// TIA Portal V20 export
TYPE "HMI_MotRevL"
   STRUCT
      FwdMan : Bool := FALSE;   // 1=Start: Forward Start Command in Manual Mode
      StopMan : Bool := FALSE;   // 1=Stop: Stop Command in Manual Mode
      RevMan : Bool := FALSE;   // 1=Start: Reverse Start Command in Manual Mode
      AutModOp : Bool := FALSE;   // 1=Auto Mode: Auto Mode by Operator
      ManModOp : Bool := TRUE;   // 1=Manual Mode: Manual Mode by Operator
      LocalLi : Bool;   // 1=Local Mode: Local Operation by Field Signal
      LocalOp : Bool := FALSE;   // 1=Local Mode: Local Operation by Operator
      OosOp : Bool := FALSE;   // 1=Oos Mode: Oos Mode by Operator
      FwdLocal : Bool;   // 1=Start Local: Field Forward Start Signal
      StopLocal : Bool;   // 1=Stop Local: Field Stop Signal
      RevLocal : Bool;   // 1=Start Local: Field Reverse Start Signal
      Monitor : Bool := TRUE;   // 1=Monitor ON, 0=Monitor OFF: Feedback Monitor
      MonTiStatic : Real := 3.0;   // Monitoring Time of Feedback [s]
      MonTiDynamic : Real := 3.0;   // Monitoring Time of Feedback on starting or on change in control output [s]
      MonTiDyStop : Real := 3.0;   // Monitoring Time of Feedback on stopping in control output [s]
      RapidStp : Bool := FALSE;   // 1 = Motor Rapid Stop command
      RstOp : Bool := FALSE;   // Operator Reset Signal
      Permit_ST : Byte := BYTE#16#FF;   // Permit Signal Status
      PermRev_ST : Byte := BYTE#16#FF;   // PermRev Signal Status
      Intlock_ST : Byte := BYTE#16#FF;   // Intlock Signal Status
      IntlRev_ST : Byte := BYTE#16#FF;   // IntlRev Signal Status
      Protect_ST : Byte := BYTE#16#FF;   // Protect Signal Status
      ProtRev_ST : Byte := BYTE#16#FF;   // ProtRev Signal Status
      UserAna1 : Real;   // User Analog Input 1
      UA1unit : Int := 0;   // Unit of UserAna1
      UserAna2 : Real;   // User Analog Input 2
      UA2unit : Int := 0;   // Unit of UserAna2
      BatchID : DWord := 16#0;   // Current Batch ID (number)
      BatchName : String[32] := '';   // Current Batch Name
      StepNo : DWord := 16#0;   // Batch Step Number
      CurrMon { ExternalWritable := 'False'} : DInt := 0;   // Remaining monitoring time [s]
      OS_PermOut { ExternalWritable := 'False'} : DWord := DWORD#16#FFFF_FFFF;   // Operator Permission: Output for OS
      OS_PermLog { ExternalWritable := 'False'} : DWord := DWORD#16#FFFF_FFFF;   // Operator Permission: Output for OS
      OpSt_Out { ExternalWritable := 'False'} : DWord := 16#0;   // Enabled operator stations
      ST_Worst { ExternalWritable := 'False'} : Byte := 16#80;   // Worst Signal Status
      AutoST { ExternalWritable := 'False'} : Byte := 16#80;   // Worst Signal Status of the automatic commands
      Status1 { ExternalWritable := 'False'} : DWord := 16#0;   // Status1 Word
      Status2 { ExternalWritable := 'False'} : DWord := 16#0;   // Status2 Word
      Status3 { ExternalWritable := 'False'} : DWord := 16#0;   // Status3 Word
      Status4 { ExternalWritable := 'False'} : DWord := 16#0;   // Status4 Word
      Status5 { ExternalWritable := 'False'} : DWord := 16#0;   // Status5 Word
      AlarmState { ExternalWritable := 'False'} : Word;   // Alarm State for group display / Alarm Status for group display
   END_STRUCT;
END_TYPE
